TYPE UnitController EXTENDS UnitBase :
STRUCT
END_STRUCT
END_TYPE

(* stored: Version 1.1.0.1, ProductVersion 3.1.4022.10
   DUT UnitController: Id {3540f8c1-cc91-4ec1-8a4f-7596595f2c82} *)
